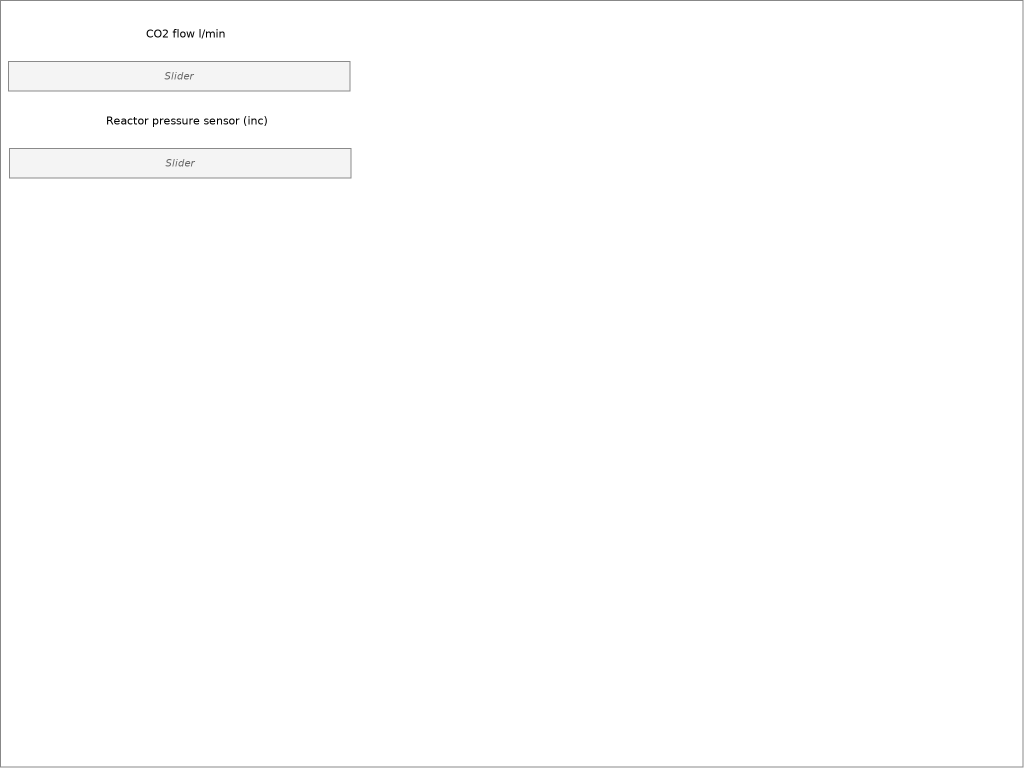
VISUALIZATION SimulationView  // 1024x768
    Slider (8,61 342x30), variable: SimulationViewBindings.flowSlider_Variable, scale 0..35
    Label (111,19 150x30), "CO2 flow l/min"
    Slider (9,148 342x30), variable: SimulationViewBindings.pressureSlider_Variable, scale 0..10000
    Label (112,106 150x30), "Reactor pressure sensor (inc)"
END_VISUALIZATION

(* stored: Version 1.1.0.1, ProductVersion 3.1.4024.9
   Visu SimulationView: Id {b2720d7c-ffee-4d76-acd0-af040e2827c5} *)
